// Mitsubishi GX Works2 project: AGV PLC Test   PLC: Q03UD

PROGRAM MAIN
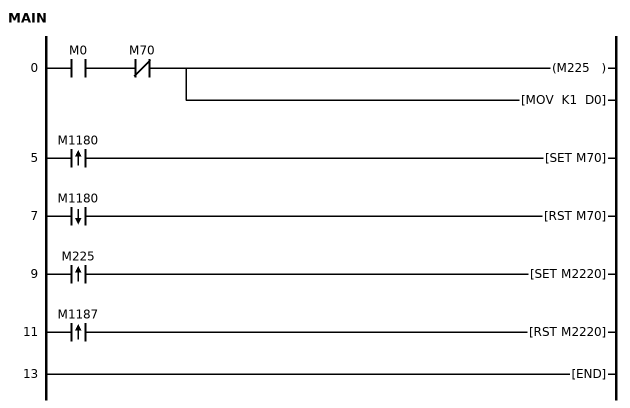
0     LD      M0
      ANI     M70
      OUT     M225
      MOV     K1 D0
5     LDP     M1180
      SET     M70
7     LDF     M1180
      RST     M70
9     LDP     M225
      SET     M2220
11    LDP     M1187
      RST     M2220
13    END
END_PROGRAM
